PROGRAM Intfc_Downstream_ML
VAR
END_VAR

// NETWORK 1

END_PROGRAM

(* stored: Version 1.1.0.1, ProductVersion 3.1.4022.11
   POU Intfc_Downstream_ML: Id {0e623b68-e6e4-425e-ad28-15fd7b9483e8}, SpecialFunc None *)
